FUNCTION_BLOCK ILOCK_BLOCK (* Prioritizes the first active input. Any subsequent conflicting signals are completely ignored until the initial input is released. *)
  (* Standard: 61499-2; Description: Copyright (c) 2023 HR Agrartechnik GmbH This program and the accompanying materials are made available under the terms of the Eclipse Public License 2.0 which is available at https://www.eclipse.org/legal/epl-2.0/ SPDX-License-Identifier: EPL-2.0 *)
  (* Version 1.0, 2026-02-23, Franz Höpfinger, HR Agrartechnik GmbH, initial API and implementation and/or initial documentation *)
  PACKAGE logiBUS::signalprocessing::interlock;
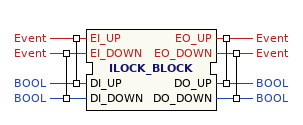
  EVENT_INPUT
    EI_UP WITH DI_UP;
    EI_DOWN WITH DI_DOWN;
  END_EVENT
  EVENT_OUTPUT
    EO_UP WITH DO_UP;
    EO_DOWN WITH DO_DOWN;
  END_EVENT
  VAR_INPUT
    DI_UP : BOOL; (* TRUE = forward, up, right, clockwise *)
    DI_DOWN : BOOL; (* TRUE = backward, down, left, counter-clockwise *)
  END_VAR
  VAR_OUTPUT
    DO_UP : BOOL; (* TRUE = forward, up, right, clockwise *)
    DO_DOWN : BOOL; (* TRUE = backward, down, left, counter-clockwise *)
  END_VAR
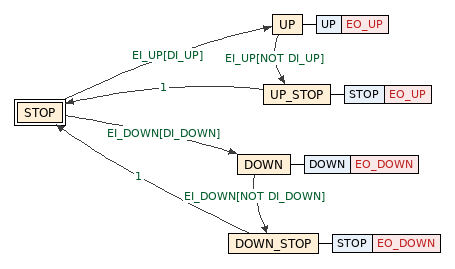
  EC_STATES
    STOP;
    UP : UP -> EO_UP;
    DOWN : DOWN -> EO_DOWN;
    UP_STOP : STOP -> EO_UP;
    DOWN_STOP : STOP -> EO_DOWN;
  END_STATES
  EC_TRANSITIONS
    STOP TO DOWN := EI_DOWN[DI_DOWN];
    STOP TO UP := EI_UP[DI_UP];
    DOWN TO DOWN_STOP := EI_DOWN[NOT DI_DOWN];
    UP TO UP_STOP := EI_UP[NOT DI_UP];
    DOWN_STOP TO STOP := 1;
    UP_STOP TO STOP := 1;
  END_TRANSITIONS
  ALGORITHM UP IN ST:
DO_UP := BOOL#TRUE;
DO_DOWN := BOOL#FALSE;
  END_ALGORITHM
  ALGORITHM DOWN IN ST:
DO_UP := BOOL#FALSE;
DO_DOWN := BOOL#TRUE;
  END_ALGORITHM
  ALGORITHM STOP IN ST:
DO_UP := BOOL#FALSE;
DO_DOWN := BOOL#FALSE;
  END_ALGORITHM
END_FUNCTION_BLOCK
